// TIA Portal project "FactoryIO_Template_S7-1200_V16_V16" (V16)
// Vorlageprojekt für das Buch mit Zielsystem S7-1200

(* hardware
DEVICE "S7-1200-Station_1"  S7-1200 Station
   slot 0: "Baugruppenträger_0"  Rack  V1.0
   slot 1: "PLC_1"  CPU 1211C DC/DC/DC  6ES7 211-1AE40-0XB0  V4.1
*)

// ===== PLC "PLC_1"  CPU 1211C DC/DC/DC =====

VAR_GLOBAL   // PLC tag table "Standard-Variablentabelle"
   "START" AT %I0.0 : Bool;
   "STOP" AT %I0.1 : Bool;
   "RESET" AT %I0.2 : Bool;
   "MEDUIM" AT %I0.3 : Bool;
   "LARGE" AT %I0.4 : Bool;
   "AT 0" AT %I0.5 : Bool;
   "AT 2 LOW" AT %I0.6 : Bool;
   "AT 2 HIGH" AT %I0.7 : Bool;
   "AT 3 LOW" AT %I1.0 : Bool;
   "AT 3 HIGH" AT %I1.1 : Bool;
   "R LIMIT" AT %I1.2 : Bool;
   "ENTRY 1" AT %I1.3 : Bool;
   "ENTRY 2" AT %I1.4 : Bool;
   "CONVEYOR 0" AT %Q0.0 : Bool;
   "CONVEYOR 1" AT %Q0.1 : Bool;
   "CONVEYOR 2" AT %Q0.2 : Bool;
   "LOAD" AT %Q0.3 : Bool;
   "UNLOAD" AT %Q0.4 : Bool;
   "UP" AT %Q0.5 : Bool;
   "DOWN" AT %Q0.6 : Bool;
   "SLOW" AT %Q0.7 : Bool;
   "M1" AT %M0.0 : Bool;
   "M2" AT %M0.1 : Bool;
   "M3" AT %M0.2 : Bool;
   "M4" AT %M0.3 : Bool;
   "M5" AT %M0.4 : Bool;
   "M6" AT %M0.5 : Bool;
   "M7" AT %M0.6 : Bool;
END_VAR

// folder: System blocks/Program resources

DATA_BLOCK "c1'"   // DB1
{ S7_Optimized_Access := 'TRUE' }
AUTHOR : Simatic
FAMILY : IEC
NAME : CNTR
VERSION : 1.0
// stored: InstanceOfName IEC_COUNTER
"IEC_COUNTER"
BEGIN
END_DATA_BLOCK

// folder: (top level)

FUNCTION "MHJ-PLC-Lab-Function-S71200" : Void   // FC9000, SCL
{ S7_Optimized_Access := 'TRUE' }
VERSION : 0.1
   VAR_TEMP
      rdTimeReturn : Int;
      outputTime : DTL;
      SyncVal : Byte;
      forVal : Int;
      forVal_2 : Int;
      Value : Byte;
   END_VAR
   VAR CONSTANT
      CompVal : Byte := 16#34;
      Value_01 : Byte := 16#11;
      Value_01_DW : DWord := 16#A165_D992;
      Value_02_DW : DWord := 16#58BE_4401;
   END_VAR
BEGIN

   #Value:=PEEK(area := 16#82,
        dbNumber := 0,
        byteOffset := 511);
   #Value := #Value + 1;

   POKE(area := 16#82,
        dbNumber := 0,
        byteOffset := 511,
        value := #Value);

   POKE(area:=16#81,
        dbNumber:=0,
        byteOffset:=1016,
        value:=#Value_01_DW);
   POKE(area := 16#81,
        dbNumber := 0,
        byteOffset := 1020,
        value := #Value_02_DW);

   POKE(area := 16#81,
        dbNumber := 0,
        byteOffset := 511,
        value := B#16#00);

   FOR #forVal := 0 TO 120 DO
       FOR #forVal_2:=0 TO 10 DO
           #rdTimeReturn:=RD_SYS_T(#outputTime);
           #rdTimeReturn := WR_SYS_T(#outputTime);
           #rdTimeReturn := RD_SYS_T(#outputTime);
           #rdTimeReturn := WR_SYS_T(#outputTime);
       END_FOR;
       #SyncVal:= PEEK(area := 16#81,
                      dbNumber := 0,
                      byteOffset := 511);
       IF #SyncVal = #CompVal THEN
          GOTO M_1;
       END_IF;
   END_FOR;
   RETURN;

   M_1:
   POKE(area := 16#81,
        dbNumber := 0,
        byteOffset := 511,
        value := B#16#0);
END_FUNCTION

ORGANIZATION_BLOCK "Main"   // OB1, LAD, ProgramCycle
TITLE = "Main Program Sweep (Cycle)"
{ S7_Optimized_Access := 'TRUE' }
VERSION : 0.1
   VAR_INPUT
      Initial_Call : Bool;   // Initial call of this OB
      Remanence : Bool;   // =True, if remanent data are available
   END_VAR
   VAR_TEMP   // added for the SCL form of the ladder/FBD networks
      _w1 : Bool;
      _w2 : Bool;
   END_VAR
BEGIN

REGION Network 1: Konnektierungsbaustein für PLC-Lab
   // Im Netzwerk 1 wird der Konnektierungsbaustein für PLC-Lab aufgerufen.
   // Dieser Aufruf darf nicht entfernt werden!
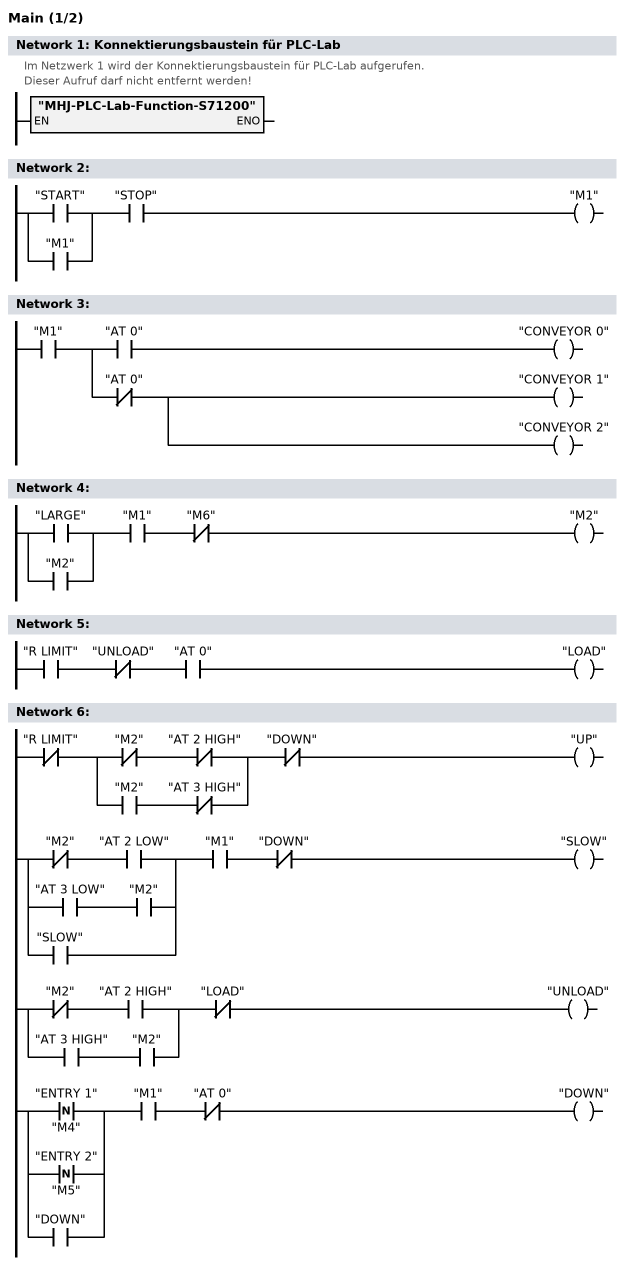
   RUNG wire#powerrail
      "MHJ-PLC-Lab-Function-S71200"()
   END_RUNG
   // the same network as SCL:
   "MHJ-PLC-Lab-Function-S71200"();
END_REGION

REGION Network 2
   RUNG wire#powerrail
      Contact( "START" )
      wire#w1
      Contact( "STOP" )
      Coil( "M1" )
   END_RUNG
   RUNG wire#powerrail
      Contact( "M1" )
   END_RUNG wire#w1
   // the same network as SCL:
   "M1" := ("START" OR "M1") AND "STOP";
END_REGION

REGION Network 3
   RUNG wire#powerrail
      Contact( "M1" )
      wire#w1
      Contact( "AT 0" )
      Coil( "CONVEYOR 0" )
   END_RUNG
   RUNG wire#w1
      I_Contact( "AT 0" )
      wire#w2
      Coil( "CONVEYOR 1" )
   END_RUNG
   RUNG wire#w2
      Coil( "CONVEYOR 2" )
   END_RUNG
   // the same network as SCL:
   "CONVEYOR 0" := "M1" AND "AT 0";
   "CONVEYOR 1" := "M1" AND NOT "AT 0";
   "CONVEYOR 2" := "CONVEYOR 1";
END_REGION

REGION Network 4
   RUNG wire#powerrail
      Contact( "LARGE" )
      wire#w1
      Contact( "M1" )
      I_Contact( "M6" )
      Coil( "M2" )
   END_RUNG
   RUNG wire#powerrail
      Contact( "M2" )
   END_RUNG wire#w1
   // the same network as SCL:
   "M2" := ("LARGE" OR "M2") AND "M1" AND NOT "M6";
END_REGION

REGION Network 5
   RUNG wire#powerrail
      Contact( "R LIMIT" )
      I_Contact( "UNLOAD" )
      Contact( "AT 0" )
      Coil( "LOAD" )
   END_RUNG
   // the same network as SCL:
   "LOAD" := "R LIMIT" AND NOT "UNLOAD" AND "AT 0";
END_REGION

REGION Network 6
   RUNG wire#powerrail
      I_Contact( "R LIMIT" )
      wire#w1
      I_Contact( "M2" )
      I_Contact( "AT 2 HIGH" )
      wire#w2
      I_Contact( "DOWN" )
      Coil( "UP" )
   END_RUNG
   RUNG wire#w1
      Contact( "M2" )
      I_Contact( "AT 3 HIGH" )
   END_RUNG wire#w2
   RUNG wire#powerrail
      I_Contact( "M2" )
      Contact( "AT 2 LOW" )
      wire#w3
      Contact( "M1" )
      I_Contact( "DOWN" )
      Coil( "SLOW" )
   END_RUNG
   RUNG wire#powerrail
      Contact( "AT 3 LOW" )
      Contact( "M2" )
   END_RUNG wire#w3
   RUNG wire#powerrail
      Contact( "SLOW" )
   END_RUNG wire#w3
   RUNG wire#powerrail
      I_Contact( "M2" )
      Contact( "AT 2 HIGH" )
      wire#w4
      I_Contact( "LOAD" )
      Coil( "UNLOAD" )
   END_RUNG
   RUNG wire#powerrail
      Contact( "AT 3 HIGH" )
      Contact( "M2" )
   END_RUNG wire#w4
   RUNG wire#powerrail
      N_Contact(operand := "ENTRY 1", bit := "M4")
      wire#w5
      Contact( "M1" )
      I_Contact( "AT 0" )
      Coil( "DOWN" )
   END_RUNG
   RUNG wire#powerrail
      N_Contact(operand := "ENTRY 2", bit := "M5")
   END_RUNG wire#w5
   RUNG wire#powerrail
      Contact( "DOWN" )
   END_RUNG wire#w5
   // the same network as SCL:
   "UP" := NOT "R LIMIT" AND ((NOT "M2" AND NOT "AT 2 HIGH") OR ("M2" AND NOT "AT 3 HIGH")) AND NOT "DOWN";
   "SLOW" := ((NOT "M2" AND "AT 2 LOW") OR ("AT 3 LOW" AND "M2") OR "SLOW") AND "M1" AND NOT "DOWN";
   "UNLOAD" := ((NOT "M2" AND "AT 2 HIGH") OR ("AT 3 HIGH" AND "M2")) AND NOT "LOAD";
   #_w1 := NOT "ENTRY 1" AND "M4";   // falling edge of "ENTRY 1"
   "M4" := "ENTRY 1";
   #_w2 := NOT "ENTRY 2" AND "M5";   // falling edge of "ENTRY 2"
   "M5" := "ENTRY 2";
   "DOWN" := (#_w1 OR #_w2 OR "DOWN") AND "M1" AND NOT "AT 0";
END_REGION

REGION Network 7
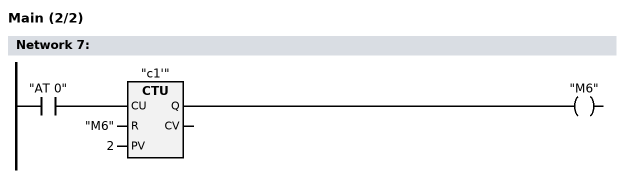
   "c1'".CTU(CU := "AT 0", R := "M6", PV := 2);
   "M6" := "c1'".Q;
END_REGION
END_ORGANIZATION_BLOCK